FUNCTION "FC2039_ZC_TQ" : Void
TITLE = FC2038_TQ
{ S7_Optimized_Access := 'TRUE' }
AUTHOR : HCR
FAMILY : ZeusControl
VERSION : 1.0
//Funcion para gestion dispositivo tanque.
   VAR_INPUT
      Pulso1seg : Bool;
      Arranque : Bool;
   END_VAR

   VAR_TEMP
      for_i : Int;
      for_mux_cambios : Int;
      for_mux : Int;
      t_Index : Int;
      t_oldIndex : Int;
      t_NumLL : Int;
      t_NumHL : Int;
      t_NumBH : Int;
      t_NumNivel : Int;
      t_NumTemperatura : Int;
      t_x0 : Real;
      t_x1 : Real;
      t_x : Real;
      t_y0 : Real;
      t_y1 : Real;
      t_RadioCilindro : Real;
      t_RadioConoInf : Real;
      t_RadioActual : Real;
      t_Vol1 : Real;
      t_Vol2 : Real;
      t_Vol3 : Real;
      t_ConsignaAgitador : Real;
      t_AlarmaNivel : Bool;
      t_AlarmaTemperatura : Bool;
      t_VacioLL : Bool;
      t_VacioEA : Bool;
      t_AlarmaConfigD : Bool;
      t_AlarmaConfigEA : Bool;
      t_AlarmaConfigV : Bool;
      t_AlarmaConfigAG : Bool;
      t_HistPositiva : Real;
      t_HistNegativa : Real;
      t_ElseCase : Bool;
   END_VAR

   VAR CONSTANT
      CONSTANTE_EMPIRICA : Real := 10.1;
      CONSTANTE_PI : Real := 3.141593;
      ESTADO_DESHABILITADO : Int := 0;
      ESTADO_SUCIO : Int := 1;
      ESTADO_LIMPIO : Int := 2;
      ESTADO_PRODUCTO : Int := 3;
      ESTADO_CIP : Int := 4;
   END_VAR


BEGIN
	(*
	ZEUS CONTROL, S.A.
	(c)Copyright (2022) All Rights Reserved
	--------------------------------------------------------------------------------------

	Software:       TIA Portal 16
	Restricciones:  PLC serie 1200/1500

	Nombre:         DISPOSITIVO TANQUE
	Descripcion:    Modelo de dispositivo tanque

	Dependencias:
	    FC:         FC15025_ZC_CONTADOR_TIEMPO_V1_01
	    FB:         -
	    DB:         DB2018_DISP_TQ
	                DB1_SYS
	    UDT:        ZC_DISP_TQ
	                ZC_MUX
	                ZC_TON
	                ZC_CONTADOR_TIEMPO

	Change log:

	    Version     Fecha       Tecnico a cargo     Descripción

	    01.00.01    26.04.2022  (HCR)               Primera versión.
	    01.00.02    09.10.2023  (HCR)               Cambio en activacion dispositivos para que actue solamente cuando tenga producto.
	    01.00.03    15.04.2024  (ABH)               Se añade gestion multiplexado para Scada (no indexado)
	    01.00.04    08.01.2025  (ABH)               Se añade entrada de primer arranque del PLC para resetear indices de multiplexado
	                                                Se añade movimiento de TQ[0] a multiplexado en caso de que el indice sea 0.
	    01.00.05    24.01.2025  (ABH)               Se modifica la logica del multiplexado, la asignacion de oldindex se cambia de sitio ya que de vez en cuando (dependiendo de cuando el HMI
	                                                realiza la comunicacion asincrona con el PLC) no detectaba el cambio y se machacaban valores.
	    01.00.16    26.03.2025  (ABH)               Se añade variable grupo de alarma para separar los nuevos avisos por cuadro.
	    02.00.00    17.12.2025  (ABH)               Se eliminan los idiomas. Se utiliza codigos para trazabilidad. Se elimina entrada "Idioma". Se elimina nombre de UDT. Se añade indexHMI para lista de
	                                                texto en sistemas de supervision.

	//=====================================================================================
	*)

	REGION MULTIPLEXADO

	    //  ===========================================================================================================
	    //  Al arranque del PLC, ponemos a 0 todos los indices de los multiplexados y salimos del bloque sin gestionarlo
	    IF #Arranque THEN
	        FOR #for_mux := 0 TO "N_MAX_MUX_DISP" DO
	            "DB2039_TQ".Mux[#for_mux].Index :=
	            "DB2039_TQ".Mux[#for_mux].oldIndex := 0;
	        END_FOR;
	        RETURN;
	    END_IF;

	    //  ===========================================================================================================
	    //  Gestion de multiplexado
	    FOR #for_mux := 0 TO "N_MAX_MUX_DISP" DO

	        //  ===============================================================================================================
	        //  Antes de iniciar la logica del multiplexado, revisamos los limites
	        REGION LIMITES

	            //  ===========================================================================================================
	            //  Limites
	            IF "DB2039_TQ".Mux[#for_mux].Index < 0 THEN
	                "DB2039_TQ".Mux[#for_mux].Index := 0;
	            END_IF;
	            IF "DB2039_TQ".Mux[#for_mux].Index > "N_MAX_DISP_TQ" THEN
	                "DB2039_TQ".Mux[#for_mux].Index := "N_MAX_DISP_TQ";
	            END_IF;
	            IF "DB2039_TQ".Mux[#for_mux].Index >= "N_MAX_DISP_TQ" THEN
	                "DB2039_TQ".Mux[#for_mux].MaxVisible := TRUE;
	            ELSE
	                "DB2039_TQ".Mux[#for_mux].MaxVisible := FALSE;
	            END_IF;

	        END_REGION

	        //  Pasamos el indice a variable temporal para evisar cambios no deseados
	        #t_Index := "DB2039_TQ".Mux[#for_mux].Index;
	        #t_oldIndex := "DB2039_TQ".Mux[#for_mux].oldIndex;

	        //  ===========================================================================================================
	        //  Valor anterior del indice
	        "DB2039_TQ".Mux[#for_mux].oldIndex := #t_Index;

	        IF "DB2039_TQ".Mux[#for_mux].Habilitar THEN

	            //  ===========================================================================================================
	            //  Gestionamos solo los tipos
	            IF #t_Index > 0 THEN



	                REGION CARGA_INICIAL

	                    //  ===========================================================================================================
	                    //  Al detectar un cambio en el indice del dispositivo, cargamos los valores del dispositivo que tenga el indice.
	                    IF #t_Index <> #t_oldIndex THEN
	                        "DB2039_TQ".Mux[#for_mux].TQ := "DB2039_TQ".TQ[#t_Index];
	                    END_IF;

	                END_REGION



	                REGION DATOS_LECTURA

	                    //  ===========================================================================================================
	                    //  Movimiento de datos gestionados en FC
	                    "DB2039_TQ".Mux[#for_mux].TQ.Hmi_Index := "DB2039_TQ".TQ[#t_Index].Hmi_Index;
	                    "DB2039_TQ".Mux[#for_mux].TQ.Hmi_Estado := "DB2039_TQ".TQ[#t_Index].Hmi_Estado;
	                    "DB2039_TQ".Mux[#for_mux].TQ.Estado_TanqueVacio  := "DB2039_TQ".TQ[#t_Index].Estado_TanqueVacio;
	                    "DB2039_TQ".Mux[#for_mux].TQ.Estado_PocisionAltura  := "DB2039_TQ".TQ[#t_Index].Estado_PocisionAltura;
	                    "DB2039_TQ".Mux[#for_mux].TQ.Estado_NivelBajo  := "DB2039_TQ".TQ[#t_Index].Estado_NivelBajo;
	                    "DB2039_TQ".Mux[#for_mux].TQ.Estado_NivelAlto  := "DB2039_TQ".TQ[#t_Index].Estado_NivelAlto;
	                    "DB2039_TQ".Mux[#for_mux].TQ.Estado_BocaHombre  := "DB2039_TQ".TQ[#t_Index].Estado_BocaHombre;
	                    "DB2039_TQ".Mux[#for_mux].TQ.Estado_Mezcla  := "DB2039_TQ".TQ[#t_Index].Estado_Mezcla;
	                    "DB2039_TQ".Mux[#for_mux].TQ.Alarmas_NivelBajo  := "DB2039_TQ".TQ[#t_Index].Alarmas_NivelBajo;
	                    "DB2039_TQ".Mux[#for_mux].TQ.Alarmas_NivelAlto  := "DB2039_TQ".TQ[#t_Index].Alarmas_NivelAlto;
	                    "DB2039_TQ".Mux[#for_mux].TQ.Alarmas_BocaHombre  := "DB2039_TQ".TQ[#t_Index].Alarmas_BocaHombre;
	                    "DB2039_TQ".Mux[#for_mux].TQ.Alarmas_Instrumentacion  := "DB2039_TQ".TQ[#t_Index].Alarmas_Instrumentacion;
	                    "DB2039_TQ".Mux[#for_mux].TQ.Alarmas_Parametros  := "DB2039_TQ".TQ[#t_Index].Alarmas_Parametros;
	                    "DB2039_TQ".Mux[#for_mux].TQ.Alarmas_General  := "DB2039_TQ".TQ[#t_Index].Alarmas_General;
	                    "DB2039_TQ".Mux[#for_mux].TQ.Alarmas_Capacidad  := "DB2039_TQ".TQ[#t_Index].Alarmas_Capacidad;
	                    "DB2039_TQ".Mux[#for_mux].TQ.Aux_VisConsignaTemperatura  := "DB2039_TQ".TQ[#t_Index].Aux_VisConsignaTemperatura;
	                    "DB2039_TQ".Mux[#for_mux].TQ.Aux_PulsoAlternarAG  := "DB2039_TQ".TQ[#t_Index].Aux_PulsoAlternarAG;
	                    "DB2039_TQ".Mux[#for_mux].TQ.Aux_MemOrdenAgitador  := "DB2039_TQ".TQ[#t_Index].Aux_MemOrdenAgitador;
	                    "DB2039_TQ".Mux[#for_mux].TQ.Aux_MemOrdenTemperatura  := "DB2039_TQ".TQ[#t_Index].Aux_MemOrdenTemperatura;
	                    "DB2039_TQ".Mux[#for_mux].TQ.Aux_MemOrdenProducto  := "DB2039_TQ".TQ[#t_Index].Aux_MemOrdenProducto;
	                    "DB2039_TQ".Mux[#for_mux].TQ.Aux_MemEstadoCIP  := "DB2039_TQ".TQ[#t_Index].Aux_MemEstadoCIP;
	                    "DB2039_TQ".Mux[#for_mux].TQ.Aux_CipOK := "DB2039_TQ".TQ[#t_Index].Aux_CipOK;

	                    "DB2039_TQ".Mux[#for_mux].TQ.Orden_ParoControlAgitador := "DB2039_TQ".TQ[#t_Index].Orden_ParoControlAgitador;
	                    "DB2039_TQ".Mux[#for_mux].TQ.Orden_ParoControlTemp := "DB2039_TQ".TQ[#t_Index].Orden_ParoControlTemp;

	                    "DB2039_TQ".Mux[#for_mux].TQ.Estado_EA_Nivel  := "DB2039_TQ".TQ[#t_Index].Estado_EA_Nivel;
	                    "DB2039_TQ".Mux[#for_mux].TQ.Estado_EA_Temperatura  := "DB2039_TQ".TQ[#t_Index].Estado_EA_Temperatura;
	                    "DB2039_TQ".Mux[#for_mux].TQ.Estado_Tanque := "DB2039_TQ".TQ[#t_Index].Estado_Tanque;
	                    "DB2039_TQ".Mux[#for_mux].TQ.Estado_Producto1  := "DB2039_TQ".TQ[#t_Index].Estado_Producto1;
	                    "DB2039_TQ".Mux[#for_mux].TQ.Estado_Producto2  := "DB2039_TQ".TQ[#t_Index].Estado_Producto2;
	                    "DB2039_TQ".Mux[#for_mux].TQ.Estado_Volumen  := "DB2039_TQ".TQ[#t_Index].Estado_Volumen;
	                    "DB2039_TQ".Mux[#for_mux].TQ.Estado_Presion  := "DB2039_TQ".TQ[#t_Index].Estado_Presion;
	                    "DB2039_TQ".Mux[#for_mux].TQ.Estado_Altura  := "DB2039_TQ".TQ[#t_Index].Estado_Altura;

	                    "DB2039_TQ".Mux[#for_mux].TQ.Tiempos_TiempoProducto := "DB2039_TQ".TQ[#t_Index].Tiempos_TiempoProducto;
	                    "DB2039_TQ".Mux[#for_mux].TQ.Tiempos_TiempoLimpio := "DB2039_TQ".TQ[#t_Index].Tiempos_TiempoLimpio;
	                    "DB2039_TQ".Mux[#for_mux].TQ.Tiempos_RetTanqueVacio  := "DB2039_TQ".TQ[#t_Index].Tiempos_RetTanqueVacio;
	                    "DB2039_TQ".Mux[#for_mux].TQ.Tiempos_AgitadorONActual := "DB2039_TQ".TQ[#t_Index].Tiempos_AgitadorONActual;
	                    "DB2039_TQ".Mux[#for_mux].TQ.Tiempos_AgitadorOFFActual := "DB2039_TQ".TQ[#t_Index].Tiempos_AgitadorOFFActual;

	                    "DB2039_TQ".Mux[#for_mux].TQ.Config_HabilitarCalculoVol := "DB2039_TQ".TQ[#t_Index].Config_HabilitarCalculoVol;
	                    "DB2039_TQ".Mux[#for_mux].TQ.Config_HabilitarCamisa := "DB2039_TQ".TQ[#t_Index].Config_HabilitarCamisa;
	                    "DB2039_TQ".Mux[#for_mux].TQ.Config_HabilitarAlarmas := "DB2039_TQ".TQ[#t_Index].Config_HabilitarAlarmas;
	                    "DB2039_TQ".Mux[#for_mux].TQ.Config_HabilitarAgitador := "DB2039_TQ".TQ[#t_Index].Config_HabilitarAgitador;
	                    "DB2039_TQ".Mux[#for_mux].TQ.Config_GrupoAlarma := "DB2039_TQ".TQ[#t_Index].Config_GrupoAlarma;

	                    "DB2039_TQ".Mux[#for_mux].TQ.Aux_ValorTarjetaNivel  := "DB2039_TQ".TQ[#t_Index].Aux_ValorTarjetaNivel;
	                    "DB2039_TQ".Mux[#for_mux].TQ.Aux_ValorIngeneriaTemperatura  := "DB2039_TQ".TQ[#t_Index].Aux_ValorIngeneriaTemperatura;
	                    "DB2039_TQ".Mux[#for_mux].TQ.Orden_Temperatura := "DB2039_TQ".TQ[#t_Index].Orden_Temperatura;
	                    "DB2039_TQ".Mux[#for_mux].TQ.Orden_Agitacion := "DB2039_TQ".TQ[#t_Index].Orden_Agitacion;
	                    "DB2039_TQ".Mux[#for_mux].TQ.Orden_CIP := "DB2039_TQ".TQ[#t_Index].Orden_CIP;
	                    "DB2039_TQ".Mux[#for_mux].TQ.Orden_Producto := "DB2039_TQ".TQ[#t_Index].Orden_Producto;
	                    "DB2039_TQ".Mux[#for_mux].TQ.Orden_TipoProducto := "DB2039_TQ".TQ[#t_Index].Orden_TipoProducto;
	                    "DB2039_TQ".Mux[#for_mux].TQ.Orden_ConsignaAgitador := "DB2039_TQ".TQ[#t_Index].Orden_ConsignaAgitador;

	                END_REGION

	                REGION DATOS_ESCRITURA

	                    //  ===========================================================================================================
	                    //  Reinicializamos valor existe cambio
	                    "DB2039_TQ".Mux[#for_mux].ExisteCambio := false;

	                    //  ===========================================================================================================
	                    //  Ordenes
	                    IF "DB2039_TQ".Mux[#for_mux].TQ.Estado_TanqueNuevo <> "DB2039_TQ".TQ[#t_Index].Estado_TanqueNuevo THEN
	                        "DB2039_TQ".TQ[#t_Index].Estado_TanqueNuevo := "DB2039_TQ".Mux[#for_mux].TQ.Estado_TanqueNuevo;
	                        "DB2039_TQ".Mux[#for_mux].ExisteCambio := true;
	                    END_IF;
	                    IF "DB2039_TQ".Mux[#for_mux].TQ.Estado_ProductoNuevo <> "DB2039_TQ".TQ[#t_Index].Estado_ProductoNuevo THEN
	                        "DB2039_TQ".TQ[#t_Index].Estado_ProductoNuevo := "DB2039_TQ".Mux[#for_mux].TQ.Estado_ProductoNuevo;
	                        "DB2039_TQ".Mux[#for_mux].ExisteCambio := true;
	                    END_IF;
	                    IF "DB2039_TQ".Mux[#for_mux].TQ.Orden_CambioEstado <> "DB2039_TQ".TQ[#t_Index].Orden_CambioEstado THEN
	                        "DB2039_TQ".TQ[#t_Index].Orden_CambioEstado := "DB2039_TQ".Mux[#for_mux].TQ.Orden_CambioEstado;
	                        "DB2039_TQ".Mux[#for_mux].TQ.Orden_CambioEstado := FALSE;
	                        "DB2039_TQ".Mux[#for_mux].ExisteCambio := true;
	                     END_IF;
	                    IF "DB2039_TQ".Mux[#for_mux].TQ.Orden_CambioProd1 <> "DB2039_TQ".TQ[#t_Index].Orden_CambioProd1 THEN
	                        "DB2039_TQ".TQ[#t_Index].Orden_CambioProd1 := "DB2039_TQ".Mux[#for_mux].TQ.Orden_CambioProd1;
	                        "DB2039_TQ".Mux[#for_mux].TQ.Orden_CambioProd1 := FALSE;
	                        "DB2039_TQ".Mux[#for_mux].ExisteCambio := true;
	                    END_IF;
	                    IF "DB2039_TQ".Mux[#for_mux].TQ.Orden_CambioProd2 <> "DB2039_TQ".TQ[#t_Index].Orden_CambioProd2 THEN
	                        "DB2039_TQ".TQ[#t_Index].Orden_CambioProd2 := "DB2039_TQ".Mux[#for_mux].TQ.Orden_CambioProd2;
	                        "DB2039_TQ".Mux[#for_mux].TQ.Orden_CambioProd2 := FALSE;
	                        "DB2039_TQ".Mux[#for_mux].ExisteCambio := true;
	                    END_IF;

	                    //  ===========================================================================================================
	                    //  Configuracion
	                    IF "DB2039_TQ".Mux[#for_mux].TQ.Config_HabilitarControlAgitacion <> "DB2039_TQ".TQ[#t_Index].Config_HabilitarControlAgitacion THEN
	                        "DB2039_TQ".TQ[#t_Index].Config_HabilitarControlAgitacion := "DB2039_TQ".Mux[#for_mux].TQ.Config_HabilitarControlAgitacion;
	                        "DB2039_TQ".Mux[#for_mux].ExisteCambio := true;
	                    END_IF;
	                    IF "DB2039_TQ".Mux[#for_mux].TQ.Config_HabilitarControlTemp <> "DB2039_TQ".TQ[#t_Index].Config_HabilitarControlTemp THEN
	                        "DB2039_TQ".TQ[#t_Index].Config_HabilitarControlTemp := "DB2039_TQ".Mux[#for_mux].TQ.Config_HabilitarControlTemp;
	                        "DB2039_TQ".Mux[#for_mux].ExisteCambio := true;
	                     END_IF;
	                    IF "DB2039_TQ".Mux[#for_mux].TQ.Config_TipoControlTemperatura <> "DB2039_TQ".TQ[#t_Index].Config_TipoControlTemperatura THEN
	                        "DB2039_TQ".TQ[#t_Index].Config_TipoControlTemperatura := "DB2039_TQ".Mux[#for_mux].TQ.Config_TipoControlTemperatura;
	                        "DB2039_TQ".Mux[#for_mux].ExisteCambio := true;
	                    END_IF;
	                    IF "DB2039_TQ".Mux[#for_mux].TQ.Config_NumeroEANivel <> "DB2039_TQ".TQ[#t_Index].Config_NumeroEANivel THEN
	                        "DB2039_TQ".TQ[#t_Index].Config_NumeroEANivel := "DB2039_TQ".Mux[#for_mux].TQ.Config_NumeroEANivel;
	                        "DB2039_TQ".Mux[#for_mux].ExisteCambio := true;
	                     END_IF;
	                    IF "DB2039_TQ".Mux[#for_mux].TQ.Config_NumeroEATemp <> "DB2039_TQ".TQ[#t_Index].Config_NumeroEATemp THEN
	                        "DB2039_TQ".TQ[#t_Index].Config_NumeroEATemp := "DB2039_TQ".Mux[#for_mux].TQ.Config_NumeroEATemp;
	                        "DB2039_TQ".Mux[#for_mux].ExisteCambio := true;
	                    END_IF;
	                    IF "DB2039_TQ".Mux[#for_mux].TQ.Config_NumeroLL <> "DB2039_TQ".TQ[#t_Index].Config_NumeroLL THEN
	                        "DB2039_TQ".TQ[#t_Index].Config_NumeroLL := "DB2039_TQ".Mux[#for_mux].TQ.Config_NumeroLL;
	                        "DB2039_TQ".Mux[#for_mux].ExisteCambio := true;
	                    END_IF;
	                    IF "DB2039_TQ".Mux[#for_mux].TQ.Config_NumeroHL <> "DB2039_TQ".TQ[#t_Index].Config_NumeroHL THEN
	                        "DB2039_TQ".TQ[#t_Index].Config_NumeroHL := "DB2039_TQ".Mux[#for_mux].TQ.Config_NumeroHL;
	                        "DB2039_TQ".Mux[#for_mux].ExisteCambio := true;
	                    END_IF;
	                    IF "DB2039_TQ".Mux[#for_mux].TQ.Config_NumeroBH <> "DB2039_TQ".TQ[#t_Index].Config_NumeroBH THEN
	                        "DB2039_TQ".TQ[#t_Index].Config_NumeroBH := "DB2039_TQ".Mux[#for_mux].TQ.Config_NumeroBH;
	                        "DB2039_TQ".Mux[#for_mux].ExisteCambio := true;
	                     END_IF;
	                    IF "DB2039_TQ".Mux[#for_mux].TQ.Config_NumeroVA <> "DB2039_TQ".TQ[#t_Index].Config_NumeroVA THEN
	                        "DB2039_TQ".TQ[#t_Index].Config_NumeroVA := "DB2039_TQ".Mux[#for_mux].TQ.Config_NumeroVA;
	                        "DB2039_TQ".Mux[#for_mux].ExisteCambio := true;
	                     END_IF;
	                    IF "DB2039_TQ".Mux[#for_mux].TQ.Config_NumeroAG <> "DB2039_TQ".TQ[#t_Index].Config_NumeroAG THEN
	                        "DB2039_TQ".TQ[#t_Index].Config_NumeroAG := "DB2039_TQ".Mux[#for_mux].TQ.Config_NumeroAG;
	                        "DB2039_TQ".Mux[#for_mux].ExisteCambio := true;
	                     END_IF;
	                    IF "DB2039_TQ".Mux[#for_mux].TQ.Config_TipoAgitacionTiempo <> "DB2039_TQ".TQ[#t_Index].Config_TipoAgitacionTiempo THEN
	                        "DB2039_TQ".TQ[#t_Index].Config_TipoAgitacionTiempo := "DB2039_TQ".Mux[#for_mux].TQ.Config_TipoAgitacionTiempo;
	                        "DB2039_TQ".Mux[#for_mux].ExisteCambio := true;
	                     END_IF;
	                    IF "DB2039_TQ".Mux[#for_mux].TQ.Config_TipoAgitacionVelocidad <> "DB2039_TQ".TQ[#t_Index].Config_TipoAgitacionVelocidad THEN
	                        "DB2039_TQ".TQ[#t_Index].Config_TipoAgitacionVelocidad := "DB2039_TQ".Mux[#for_mux].TQ.Config_TipoAgitacionVelocidad;
	                        "DB2039_TQ".Mux[#for_mux].ExisteCambio := true;
	                    END_IF;
	                    IF "DB2039_TQ".Mux[#for_mux].TQ.Config_TipoAgitador <> "DB2039_TQ".TQ[#t_Index].Config_TipoAgitador THEN
	                        "DB2039_TQ".TQ[#t_Index].Config_TipoAgitador := "DB2039_TQ".Mux[#for_mux].TQ.Config_TipoAgitador;
	                        "DB2039_TQ".Mux[#for_mux].ExisteCambio := true;
	                    END_IF;
	                    IF "DB2039_TQ".Mux[#for_mux].TQ.Config_EscaladoMinTarjeta <> "DB2039_TQ".TQ[#t_Index].Config_EscaladoMinTarjeta THEN
	                        "DB2039_TQ".TQ[#t_Index].Config_EscaladoMinTarjeta := "DB2039_TQ".Mux[#for_mux].TQ.Config_EscaladoMinTarjeta;
	                        "DB2039_TQ".Mux[#for_mux].ExisteCambio := true;
	                    END_IF;
	                    IF "DB2039_TQ".Mux[#for_mux].TQ.Config_EscaladoMaxTarjeta <> "DB2039_TQ".TQ[#t_Index].Config_EscaladoMaxTarjeta THEN
	                        "DB2039_TQ".TQ[#t_Index].Config_EscaladoMaxTarjeta := "DB2039_TQ".Mux[#for_mux].TQ.Config_EscaladoMaxTarjeta;
	                        "DB2039_TQ".Mux[#for_mux].ExisteCambio := true;
	                     END_IF;
	                    IF "DB2039_TQ".Mux[#for_mux].TQ.Config_EscaladoMinIngenieria <> "DB2039_TQ".TQ[#t_Index].Config_EscaladoMinIngenieria THEN
	                        "DB2039_TQ".TQ[#t_Index].Config_EscaladoMinIngenieria := "DB2039_TQ".Mux[#for_mux].TQ.Config_EscaladoMinIngenieria;
	                        "DB2039_TQ".Mux[#for_mux].ExisteCambio := true;
	                     END_IF;
	                    IF "DB2039_TQ".Mux[#for_mux].TQ.Config_EscaladoMaxIngenieria <> "DB2039_TQ".TQ[#t_Index].Config_EscaladoMaxIngenieria THEN
	                        "DB2039_TQ".TQ[#t_Index].Config_EscaladoMaxIngenieria := "DB2039_TQ".Mux[#for_mux].TQ.Config_EscaladoMaxIngenieria;
	                        "DB2039_TQ".Mux[#for_mux].ExisteCambio := true;
	                     END_IF;
	                    IF "DB2039_TQ".Mux[#for_mux].TQ.Config_ConsignaTemperatura <> "DB2039_TQ".TQ[#t_Index].Config_ConsignaTemperatura THEN
	                        "DB2039_TQ".TQ[#t_Index].Config_ConsignaTemperatura := "DB2039_TQ".Mux[#for_mux].TQ.Config_ConsignaTemperatura;
	                        "DB2039_TQ".Mux[#for_mux].ExisteCambio := true;
	                     END_IF;
	                    IF "DB2039_TQ".Mux[#for_mux].TQ.Config_HisteresisTemperatura <> "DB2039_TQ".TQ[#t_Index].Config_HisteresisTemperatura THEN
	                        "DB2039_TQ".TQ[#t_Index].Config_HisteresisTemperatura := "DB2039_TQ".Mux[#for_mux].TQ.Config_HisteresisTemperatura;
	                        "DB2039_TQ".Mux[#for_mux].ExisteCambio := true;
	                    END_IF;
	                    IF "DB2039_TQ".Mux[#for_mux].TQ.Config_VolumenMinControlTemp <> "DB2039_TQ".TQ[#t_Index].Config_VolumenMinControlTemp THEN
	                        "DB2039_TQ".TQ[#t_Index].Config_VolumenMinControlTemp := "DB2039_TQ".Mux[#for_mux].TQ.Config_VolumenMinControlTemp;
	                        "DB2039_TQ".Mux[#for_mux].ExisteCambio := true;
	                    END_IF;
	                    IF "DB2039_TQ".Mux[#for_mux].TQ.Config_VolumenMaxControlTemp <> "DB2039_TQ".TQ[#t_Index].Config_VolumenMaxControlTemp THEN
	                        "DB2039_TQ".TQ[#t_Index].Config_VolumenMaxControlTemp := "DB2039_TQ".Mux[#for_mux].TQ.Config_VolumenMaxControlTemp;
	                        "DB2039_TQ".Mux[#for_mux].ExisteCambio := true;
	                    END_IF;
	                    IF "DB2039_TQ".Mux[#for_mux].TQ.Config_VolumenMinControlAgitador <> "DB2039_TQ".TQ[#t_Index].Config_VolumenMinControlAgitador THEN
	                        "DB2039_TQ".TQ[#t_Index].Config_VolumenMinControlAgitador := "DB2039_TQ".Mux[#for_mux].TQ.Config_VolumenMinControlAgitador;
	                        "DB2039_TQ".Mux[#for_mux].ExisteCambio := true;
	                    END_IF;
	                    IF "DB2039_TQ".Mux[#for_mux].TQ.Config_VolumenMaxControlAgitador <> "DB2039_TQ".TQ[#t_Index].Config_VolumenMaxControlAgitador THEN
	                        "DB2039_TQ".TQ[#t_Index].Config_VolumenMaxControlAgitador := "DB2039_TQ".Mux[#for_mux].TQ.Config_VolumenMaxControlAgitador;
	                        "DB2039_TQ".Mux[#for_mux].ExisteCambio := true;
	                    END_IF;
	                    IF "DB2039_TQ".Mux[#for_mux].TQ.Config_VolumenTanqueVacio <> "DB2039_TQ".TQ[#t_Index].Config_VolumenTanqueVacio THEN
	                        "DB2039_TQ".TQ[#t_Index].Config_VolumenTanqueVacio := "DB2039_TQ".Mux[#for_mux].TQ.Config_VolumenTanqueVacio;
	                        "DB2039_TQ".Mux[#for_mux].ExisteCambio := true;
	                    END_IF;
	                    IF "DB2039_TQ".Mux[#for_mux].TQ.Config_VelocidadMinAgitador <> "DB2039_TQ".TQ[#t_Index].Config_VelocidadMinAgitador THEN
	                        "DB2039_TQ".TQ[#t_Index].Config_VelocidadMinAgitador := "DB2039_TQ".Mux[#for_mux].TQ.Config_VelocidadMinAgitador;
	                        "DB2039_TQ".Mux[#for_mux].ExisteCambio := true;
	                    END_IF;
	                    IF "DB2039_TQ".Mux[#for_mux].TQ.Config_VelocidadMaxAgitador <> "DB2039_TQ".TQ[#t_Index].Config_VelocidadMaxAgitador THEN
	                        "DB2039_TQ".TQ[#t_Index].Config_VelocidadMaxAgitador := "DB2039_TQ".Mux[#for_mux].TQ.Config_VelocidadMaxAgitador;
	                        "DB2039_TQ".Mux[#for_mux].ExisteCambio := true;
	                    END_IF;
	                    IF "DB2039_TQ".Mux[#for_mux].TQ.Config_VelocidadFijaAgitador <> "DB2039_TQ".TQ[#t_Index].Config_VelocidadFijaAgitador THEN
	                        "DB2039_TQ".TQ[#t_Index].Config_VelocidadFijaAgitador := "DB2039_TQ".Mux[#for_mux].TQ.Config_VelocidadFijaAgitador;
	                        "DB2039_TQ".Mux[#for_mux].ExisteCambio := true;
	                    END_IF;
	                    IF "DB2039_TQ".Mux[#for_mux].TQ.Config_CapacidadTanque <> "DB2039_TQ".TQ[#t_Index].Config_CapacidadTanque THEN
	                        "DB2039_TQ".TQ[#t_Index].Config_CapacidadTanque := "DB2039_TQ".Mux[#for_mux].TQ.Config_CapacidadTanque;
	                        "DB2039_TQ".Mux[#for_mux].ExisteCambio := true;
	                    END_IF;
	                    IF "DB2039_TQ".Mux[#for_mux].TQ.Config_DiametroCilindro <> "DB2039_TQ".TQ[#t_Index].Config_DiametroCilindro THEN
	                        "DB2039_TQ".TQ[#t_Index].Config_DiametroCilindro := "DB2039_TQ".Mux[#for_mux].TQ.Config_DiametroCilindro;
	                        "DB2039_TQ".Mux[#for_mux].ExisteCambio := true;
	                    END_IF;
	                    IF "DB2039_TQ".Mux[#for_mux].TQ.Config_AlturaCilindro <> "DB2039_TQ".TQ[#t_Index].Config_AlturaCilindro THEN
	                        "DB2039_TQ".TQ[#t_Index].Config_AlturaCilindro := "DB2039_TQ".Mux[#for_mux].TQ.Config_AlturaCilindro;
	                        "DB2039_TQ".Mux[#for_mux].ExisteCambio := true;
	                    END_IF;
	                    IF "DB2039_TQ".Mux[#for_mux].TQ.Config_DiametroConoInferior <> "DB2039_TQ".TQ[#t_Index].Config_DiametroConoInferior THEN
	                        "DB2039_TQ".TQ[#t_Index].Config_DiametroConoInferior := "DB2039_TQ".Mux[#for_mux].TQ.Config_DiametroConoInferior;
	                        "DB2039_TQ".Mux[#for_mux].ExisteCambio := true;
	                    END_IF;
	                    IF "DB2039_TQ".Mux[#for_mux].TQ.Config_AnguloCono <> "DB2039_TQ".TQ[#t_Index].Config_AnguloCono THEN
	                        "DB2039_TQ".TQ[#t_Index].Config_AnguloCono := "DB2039_TQ".Mux[#for_mux].TQ.Config_AnguloCono;
	                        "DB2039_TQ".Mux[#for_mux].ExisteCambio := true;
	                    END_IF;
	                    IF "DB2039_TQ".Mux[#for_mux].TQ.Config_AlturaCono <> "DB2039_TQ".TQ[#t_Index].Config_AlturaCono THEN
	                        "DB2039_TQ".TQ[#t_Index].Config_AlturaCono := "DB2039_TQ".Mux[#for_mux].TQ.Config_AlturaCono;
	                        "DB2039_TQ".Mux[#for_mux].ExisteCambio := true;
	                    END_IF;

	                    //  ===========================================================================================================
	                    //  Tiempos
	                    IF "DB2039_TQ".Mux[#for_mux].TQ.Tiempos_AgitadorONConsigna <> "DB2039_TQ".TQ[#t_Index].Tiempos_AgitadorONConsigna THEN
	                        "DB2039_TQ".TQ[#t_Index].Tiempos_AgitadorONConsigna := "DB2039_TQ".Mux[#for_mux].TQ.Tiempos_AgitadorONConsigna;
	                        "DB2039_TQ".Mux[#for_mux].ExisteCambio := true;
	                    END_IF;
	                    IF "DB2039_TQ".Mux[#for_mux].TQ.Tiempos_AgitadorOFFConsigna <> "DB2039_TQ".TQ[#t_Index].Tiempos_AgitadorOFFConsigna THEN
	                        "DB2039_TQ".TQ[#t_Index].Tiempos_AgitadorOFFConsigna := "DB2039_TQ".Mux[#for_mux].TQ.Tiempos_AgitadorOFFConsigna;
	                        "DB2039_TQ".Mux[#for_mux].ExisteCambio := true;
	                    END_IF;


	                END_REGION

	                REGION GESTION_CAMBIOS

	                    //  ===========================================================================================================
	                    //  Si existe cambios en el dispositivo generados por SCADA, actualizamos los datos en el resto de multiplexados,
	                    //  en caso de que este abierto el mismo dispositivo.
	                    IF "DB2039_TQ".Mux[#for_mux].ExisteCambio THEN
	                        //  Recorremos todos los multiplexados
	                        FOR #for_mux_cambios := 0 TO "N_MAX_MUX_DISP" DO

	                            //  No miramos el multiplexado actual
	                            IF #for_mux_cambios <> #for_mux THEN

	                                //  En caso de que este seleccionado el mismo indice, movemos el dispositivo al multiplexado
	                                //  correspondiente
	                                IF #t_Index = "DB2039_TQ".Mux[#for_mux_cambios].Index THEN
	                                    "DB2039_TQ".Mux[#for_mux_cambios].TQ := "DB2039_TQ".TQ[#t_Index];
	                                END_IF;

	                            END_IF;

	                        END_FOR;
	                        "DB2039_TQ".Mux[#for_mux].ExisteCambio := FALSE;
	                    END_IF;

	                END_REGION

	            ELSE

	                //  ===========================================================================================================
	                //  En caso de que el indice sea 0, movemos el valor de la EA[0] que no se usa para escribir el index.
	                "DB2039_TQ".Mux[#for_mux].TQ := "DB2039_TQ".TQ[0];

	            END_IF;

	        ELSE

	            "DB2039_TQ".Mux[#for_mux].ExisteCambio := FALSE;
	            "DB2039_TQ".Mux[#for_mux].Index :=
	            "DB2039_TQ".Mux[#for_mux].oldIndex := 0;

	        END_IF;

	    END_FOR;

	END_REGION

	REGION LOGICA_DEL_DISPOSITIVO

	    // =============================================================================
	    // Resetear todas las alarmas para que se vuelvan a generar
	    FOR #for_i := 0 TO "N_MAX_DISP_AGRUP" DO
	        "DB2039_TQ".Agrup[#for_i].AlgunaAlarma := FALSE;
	        "DB2039_TQ".Agrup[#for_i].AlgunaEnManual := FALSE;
	    END_FOR;

	    FOR #for_i := 1 TO "N_MAX_DISP_TQ" DO

	        "DB2039_TQ".TQ[#t_Index].Hmi_Index := #for_i + "DISP_OFFSET_TQ";

	        // =============================================================================
	        //  CAMBIO DE ESTADO DESDE HMI/SCADA
	        IF "DB2039_TQ".TQ[#for_i].Orden_CambioEstado THEN
	            "DB2039_TQ".TQ[#for_i].Estado_Tanque := "DB2039_TQ".TQ[#for_i].Estado_TanqueNuevo;
	            "DB2039_TQ".TQ[#for_i].Orden_CambioEstado := FALSE;
	        END_IF;


	        "DB2039_TQ".TQ[#for_i].Config_Habilitar := ("DB2039_TQ".TQ[#for_i].Estado_Tanque <> #ESTADO_DESHABILITADO);

	        // =============================================================================
	        // DISPOSITIVO HABILITADO
	        // =============================================================================
	        IF "DB2039_TQ".TQ[#for_i].Config_Habilitar THEN

	            REGION LIMITE_GRUPO_ALARMA

	                IF "DB2039_TQ".TQ[#for_i].Config_GrupoAlarma < 0 THEN
	                    "DB2039_TQ".TQ[#for_i].Config_GrupoAlarma := 0;
	                END_IF;
	                IF "DB2039_TQ".TQ[#for_i].Config_GrupoAlarma > "N_MAX_DISP_AGRUP" THEN
	                    "DB2039_TQ".TQ[#for_i].Config_GrupoAlarma := "N_MAX_DISP_AGRUP";
	                END_IF;

	            END_REGION

	            REGION ASIGNAR_DISPOSITIVOS

	                // =============================================================================
	                //  ASIGNACION DISPOSITOS
	                #t_NumLL := "DB2039_TQ".TQ[#for_i].Config_NumeroLL;
	                #t_NumHL := "DB2039_TQ".TQ[#for_i].Config_NumeroHL;
	                #t_NumBH := "DB2039_TQ".TQ[#for_i].Config_NumeroBH;
	                #t_NumNivel := "DB2039_TQ".TQ[#for_i].Config_NumeroEANivel;
	                #t_NumTemperatura := "DB2039_TQ".TQ[#for_i].Config_NumeroEATemp;
	                // =============================================================================
	                //  DETECTOR BOCA DE HOMBRE
	                IF #t_NumBH > 0 AND #t_NumBH <= "N_MAX_DISP_ED" THEN
	                    "DB2039_TQ".TQ[#for_i].Estado_BocaHombre := "DB2000_ED".ED[#t_NumBH].Estado_Activado;
	                END_IF;
	                // =============================================================================
	                //  DETECTOR LL
	                IF #t_NumLL > 0 AND #t_NumLL <= "N_MAX_DISP_ED" THEN
	                    "DB2039_TQ".TQ[#for_i].Estado_NivelBajo := "DB2000_ED".ED[#t_NumLL].Estado_Activado;
	                END_IF;
	                // =============================================================================
	                //  DETECTOR HL
	                IF #t_NumHL > 0 AND #t_NumHL <= "N_MAX_DISP_ED" THEN
	                    "DB2039_TQ".TQ[#for_i].Estado_NivelAlto := "DB2000_ED".ED[#t_NumHL].Estado_Activado;
	                END_IF;
	                // =============================================================================
	                //  LECTURA VALOR TARJETA NIVEL
	                IF #t_NumNivel > 0 AND #t_NumNivel <= "N_MAX_DISP_EA" THEN
	                    "DB2039_TQ".TQ[#for_i].Aux_ValorTarjetaNivel := "DB2001_EA".EA[#t_NumNivel].Estado_ValorTarjeta;
	                END_IF;
	                // =============================================================================
	                //  LECTURA VALOR INGENERIA TEMPERATURA
	                IF #t_NumTemperatura > 0 AND #t_NumTemperatura <= "N_MAX_DISP_EA" THEN
	                    "DB2039_TQ".TQ[#for_i].Aux_ValorIngeneriaTemperatura := "DB2001_EA".EA[#t_NumTemperatura].Estado_ValorIngenieria;
	                END_IF;

	            END_REGION

	            REGION ALARMAS
	                // =============================================================================
	                //  ALARMA CONFIGURACIÓN
	                #t_AlarmaConfigD := ("DB2039_TQ".TQ[#for_i].Config_NumeroBH > "N_MAX_DISP_ED") OR ("DB2039_TQ".TQ[#for_i].Config_NumeroLL > "N_MAX_DISP_ED") OR ("DB2039_TQ".TQ[#for_i].Config_NumeroHL > "N_MAX_DISP_ED");
	                #t_AlarmaConfigEA := ("DB2039_TQ".TQ[#for_i].Config_NumeroEANivel > "N_MAX_DISP_EA") OR ("DB2039_TQ".TQ[#for_i].Config_NumeroEATemp > "N_MAX_DISP_EA");
	                #t_AlarmaConfigV := "DB2039_TQ".TQ[#for_i].Config_HabilitarCamisa AND "DB2039_TQ".TQ[#for_i].Config_NumeroVA > "N_MAX_DISP_V";

	                IF "DB2039_TQ".TQ[#for_i].Config_HabilitarAgitador THEN
	                    CASE "DB2039_TQ".TQ[#for_i].Config_TipoAgitador OF
	                        0:  // Motor
	                            #t_AlarmaConfigAG := "DB2039_TQ".TQ[#for_i].Config_NumeroAG > "N_MAX_DISP_M";
	                        1:  // VF
	                            #t_AlarmaConfigAG := "DB2039_TQ".TQ[#for_i].Config_NumeroAG > "N_MAX_DISP_M_VF";
	                            ;
	                        2:  // SINA
	                            #t_AlarmaConfigAG := "DB2039_TQ".TQ[#for_i].Config_NumeroAG > "N_MAX_DISP_M_SINA";
	                        ELSE  // Statement section ELSE
	                            #t_AlarmaConfigAG := TRUE;
	                    END_CASE;
	                END_IF;

	                "DB2039_TQ".TQ[#for_i].Alarmas_Parametros := #t_AlarmaConfigD OR #t_AlarmaConfigEA OR #t_AlarmaConfigV OR #t_AlarmaConfigAG;

	                IF "DB2039_TQ".TQ[#for_i].Config_HabilitarAlarmas THEN
	                    // =============================================================================
	                    //  ALARMA DETECTOR NIVEL MÍNIMO
	                    IF #t_NumLL > 0 AND #t_NumLL <= "N_MAX_DISP_ED" THEN
	                        "DB2039_TQ".TQ[#for_i].Alarmas_NivelBajo := NOT "DB2039_TQ".TQ[#for_i].Estado_NivelBajo;
	                    ELSE
	                        "DB2039_TQ".TQ[#for_i].Alarmas_NivelBajo := FALSE;
	                    END_IF;
	                    // =============================================================================
	                    //  ALARMA DETECTOR NIVEL MÁXIMO
	                    IF #t_NumHL > 0 AND #t_NumHL <= "N_MAX_DISP_ED" THEN
	                        "DB2039_TQ".TQ[#for_i].Alarmas_NivelAlto := "DB2039_TQ".TQ[#for_i].Estado_NivelAlto;
	                    ELSE
	                        "DB2039_TQ".TQ[#for_i].Alarmas_NivelAlto := FALSE;
	                    END_IF;
	                    // =============================================================================
	                    //  ALARMA DETECTOR BOCA HOMBRE
	                    IF #t_NumBH > 0 AND #t_NumBH <= "N_MAX_DISP_ED" THEN
	                        "DB2039_TQ".TQ[#for_i].Alarmas_BocaHombre := NOT "DB2039_TQ".TQ[#for_i].Estado_BocaHombre;
	                    ELSE
	                        "DB2039_TQ".TQ[#for_i].Alarmas_BocaHombre := FALSE;
	                    END_IF;
	                    // =============================================================================
	                    //  ALARMA DE INSTRUMENTACIÓN
	                    IF #t_NumNivel > 0 AND #t_NumNivel <= "N_MAX_DISP_EA" THEN
	                        #t_AlarmaNivel := ("DB2001_EA".EA[#t_NumNivel].Aux_Estado = 6 OR
	                        "DB2001_EA".EA[#t_NumNivel].Aux_Estado = 3 OR
	                        "DB2001_EA".EA[#t_NumNivel].Aux_Estado = 4 OR
	                        "DB2001_EA".EA[#t_NumNivel].Aux_Estado = 5 OR
	                        "DB2001_EA".EA[#t_NumNivel].Aux_Estado = 7 OR
	                        "DB2001_EA".EA[#t_NumNivel].Aux_Estado = 8);
	                    ELSE
	                        #t_AlarmaNivel := FALSE;
	                    END_IF;

	                    IF #t_NumTemperatura > 0 AND #t_NumTemperatura <= "N_MAX_DISP_EA" THEN
	                        #t_AlarmaTemperatura := ("DB2001_EA".EA[#t_NumNivel].Aux_Estado = 6 OR
	                        "DB2001_EA".EA[#t_NumTemperatura].Aux_Estado = 3 OR
	                        "DB2001_EA".EA[#t_NumTemperatura].Aux_Estado = 4 OR
	                        "DB2001_EA".EA[#t_NumTemperatura].Aux_Estado = 5 OR
	                        "DB2001_EA".EA[#t_NumTemperatura].Aux_Estado = 7 OR
	                        "DB2001_EA".EA[#t_NumTemperatura].Aux_Estado = 8);
	                    ELSE
	                        #t_AlarmaTemperatura := FALSE;
	                    END_IF;

	                    "DB2039_TQ".TQ[#for_i].Alarmas_Instrumentacion := #t_AlarmaNivel OR #t_AlarmaTemperatura OR
	                    ("DB2039_TQ".TQ[#for_i].Config_EscaladoMinIngenieria >= "DB2039_TQ".TQ[#for_i].Config_EscaladoMaxIngenieria) OR
	                    ("DB2039_TQ".TQ[#for_i].Config_EscaladoMinTarjeta >= "DB2039_TQ".TQ[#for_i].Config_EscaladoMaxTarjeta);

	                    // =============================================================================
	                    //  ALARMA POR CAPACIDAD
	                    "DB2039_TQ".TQ[#for_i].Alarmas_Capacidad := "DB2039_TQ".TQ[#for_i].Estado_Volumen > "DB2039_TQ".TQ[#for_i].Config_CapacidadTanque;

	                    // =============================================================================
	                    //  ALARMA GENERAL
	                    "DB2039_TQ".TQ[#for_i].Alarmas_General := "DB2039_TQ".TQ[#for_i].Alarmas_NivelBajo OR
	                    "DB2039_TQ".TQ[#for_i].Alarmas_NivelAlto OR
	                    "DB2039_TQ".TQ[#for_i].Alarmas_BocaHombre OR
	                    "DB2039_TQ".TQ[#for_i].Alarmas_Instrumentacion OR
	                    "DB2039_TQ".TQ[#for_i].Alarmas_Capacidad;

	                ELSE
	                    "DB2039_TQ".TQ[#for_i].Alarmas_General := FALSE;
	                    "DB2039_TQ".TQ[#for_i].Alarmas_NivelBajo := FALSE;
	                    "DB2039_TQ".TQ[#for_i].Alarmas_NivelAlto := FALSE;
	                    "DB2039_TQ".TQ[#for_i].Alarmas_BocaHombre := FALSE;
	                    "DB2039_TQ".TQ[#for_i].Alarmas_Instrumentacion := FALSE;
	                    "DB2039_TQ".TQ[#for_i].Alarmas_Capacidad := FALSE;
	                END_IF;
	            END_REGION

	            REGION VOLUMEN

	                REGION ESTADO VOLUMEN

	                    "DB2039_TQ".TQ[#for_i].Estado_EA_Nivel := 1;  //  Estado normal

	                    IF #t_NumNivel > 0 AND
	                        (("DB2039_TQ".TQ[#for_i].Config_EscaladoMaxIngenieria = "DB2039_TQ".TQ[#for_i].Config_EscaladoMinIngenieria) OR
	                        ("DB2039_TQ".TQ[#for_i].Config_EscaladoMaxTarjeta = "DB2039_TQ".TQ[#for_i].Config_EscaladoMinTarjeta) OR
	                        ("DB2001_EA".EA[#t_NumNivel].Aux_Estado = 6)) THEN
	                        "DB2039_TQ".TQ[#for_i].Estado_EA_Nivel := 6; //  Error de configuración
	                    END_IF;

	                    IF #t_NumNivel > 0 AND
	                        (("DB2039_TQ".TQ[#for_i].Config_EscaladoMaxIngenieria < "DB2039_TQ".TQ[#for_i].Config_EscaladoMinIngenieria) OR
	                        ("DB2039_TQ".TQ[#for_i].Config_EscaladoMaxTarjeta < "DB2039_TQ".TQ[#for_i].Config_EscaladoMinTarjeta) OR
	                        ("DB2001_EA".EA[#t_NumNivel].Aux_Estado = 6)) THEN
	                        "DB2039_TQ".TQ[#for_i].Estado_EA_Nivel := 6; //  Error de configuración
	                    END_IF;

	                    IF "DB2001_EA".EA[#t_NumNivel].Aux_Estado = 3 THEN
	                        "DB2039_TQ".TQ[#for_i].Estado_EA_Nivel := 3; //  Error de canal
	                    END_IF;

	                    IF "DB2001_EA".EA[#t_NumNivel].Aux_Estado = 4 THEN
	                        "DB2039_TQ".TQ[#for_i].Estado_EA_Nivel := 4; //  Volumen en alarma
	                    END_IF;

	                    IF "DB2001_EA".EA[#t_NumNivel].Aux_Estado = 5 THEN
	                        "DB2039_TQ".TQ[#for_i].Estado_EA_Nivel := 5; //  Volumen en alarma
	                    END_IF;

	                    IF "DB2001_EA".EA[#t_NumNivel].Aux_Estado = 7 THEN
	                        "DB2039_TQ".TQ[#for_i].Estado_EA_Nivel := 7; //  Error de lectura
	                    END_IF;

	                    IF "DB2001_EA".EA[#t_NumNivel].Aux_Estado = 8 THEN
	                        "DB2039_TQ".TQ[#for_i].Estado_EA_Nivel := 8; //  EA no direccionada
	                    END_IF;

	                    IF "DB2001_EA".EA[#t_NumNivel].Estado_AutoMan THEN
	                        "DB2039_TQ".TQ[#for_i].Estado_EA_Nivel := 2; //  Señal forzada
	                    END_IF;

	                    IF ("DB2001_EA".EA[#t_NumNivel].Aux_Estado = 0) OR (#t_NumNivel = 0) THEN
	                        "DB2039_TQ".TQ[#for_i].Estado_EA_Nivel := 0; //  Señal deshabilitada
	                    END_IF;

	                    // =============================================================================
	                    //  POSICIÓN DE ALTURA
	                    //  0 - Altura en cono, 1 - Altura por encima del cono
	                    "DB2039_TQ".TQ[#for_i].Estado_PocisionAltura := ("DB2039_TQ".TQ[#for_i].Estado_Altura > "DB2039_TQ".TQ[#for_i].Config_AlturaCono) AND (#t_NumNivel > 0);

	                    // =============================================================================
	                    //  TANQUE VACÍO
	                    #t_VacioLL := (NOT "DB2039_TQ".TQ[#for_i].Estado_NivelBajo) AND (#t_NumLL > 0);
	                    // =============================================================================
	                    //  GESTION TON PARA EA < VOLUMEN TANQUE VACIO
	                    //"DB2039_TQ".TQ[#for_i].Tiempos_RetTanqueVacio.SP := 10;
	                    "DB2039_TQ".TQ[#for_i].Tiempos_RetTanqueVacio.SP := 25;
	                    "DB2039_TQ".TQ[#for_i].Tiempos_RetTanqueVacio.IN := ("DB2039_TQ".TQ[#for_i].Estado_Volumen < "DB2039_TQ".TQ[#for_i].Config_VolumenTanqueVacio) AND (#t_NumNivel > 0);
	                    IF "DB2039_TQ".TQ[#for_i].Tiempos_RetTanqueVacio.IN THEN
	                        IF "DB2039_TQ".TQ[#for_i].Tiempos_RetTanqueVacio.ET >= "DB2039_TQ".TQ[#for_i].Tiempos_RetTanqueVacio.SP THEN
	                            "DB2039_TQ".TQ[#for_i].Tiempos_RetTanqueVacio.Q := TRUE;
	                        ELSE
	                            IF #Pulso1seg THEN
	                                "DB2039_TQ".TQ[#for_i].Tiempos_RetTanqueVacio.ET += 1;
	                            END_IF;
	                        END_IF;
	                    ELSE
	                        "DB2039_TQ".TQ[#for_i].Tiempos_RetTanqueVacio.ET := 0;
	                        "DB2039_TQ".TQ[#for_i].Tiempos_RetTanqueVacio.Q := FALSE;
	                    END_IF;
	                    #t_VacioEA := "DB2039_TQ".TQ[#for_i].Tiempos_RetTanqueVacio.Q;
	                    "DB2039_TQ".TQ[#for_i].Estado_TanqueVacio := #t_VacioLL OR #t_VacioEA;

	                END_REGION

	                REGION CALCULO_VOLUMEN_TANQUE

	                    // =============================================================================
	                    // HABILITADO CALCULO DE VOLUMEN
	                    IF "DB2039_TQ".TQ[#for_i].Config_HabilitarCalculoVol THEN

	                        // =============================================================================
	                        //  VALORES DE ESCALADO
	                        #t_x0 := INT_TO_REAL("DB2039_TQ".TQ[#for_i].Config_EscaladoMinTarjeta);
	                        #t_x1 := INT_TO_REAL("DB2039_TQ".TQ[#for_i].Config_EscaladoMaxTarjeta);
	                        #t_x := DINT_TO_REAL("DB2039_TQ".TQ[#for_i].Aux_ValorTarjetaNivel);
	                        #t_y0 := "DB2039_TQ".TQ[#for_i].Config_EscaladoMinIngenieria;
	                        #t_y1 := "DB2039_TQ".TQ[#for_i].Config_EscaladoMaxIngenieria;

	                        // =============================================================================
	                        // SEÑAL EN ESTADO CORRECTO
	                        IF "DB2039_TQ".TQ[#for_i].Estado_EA_Nivel <> 6 AND
	                            "DB2039_TQ".TQ[#for_i].Estado_EA_Nivel <> 3 AND
	                            "DB2039_TQ".TQ[#for_i].Estado_EA_Nivel <> 7 AND
	                            "DB2039_TQ".TQ[#for_i].Estado_EA_Nivel <> 8 THEN

	                            // =============================================================================
	                            // SEÑAL EN AUTOMATICO
	                            IF NOT "DB2001_EA".EA[#t_NumNivel].Estado_AutoMan THEN

	                                // =============================================================================
	                                // ESCALADO
	                                "DB2039_TQ".TQ[#for_i].Estado_Presion := (((#t_x - #t_x0) * ((#t_y1 - #t_y0) / (#t_x1 - #t_x0))) + #t_y0);
	                                // =============================================================================
	                                // LÍMITE MAX
	                                IF "DB2039_TQ".TQ[#for_i].Estado_Presion > "DB2039_TQ".TQ[#for_i].Config_EscaladoMaxIngenieria THEN
	                                    "DB2039_TQ".TQ[#for_i].Estado_Presion := "DB2039_TQ".TQ[#for_i].Config_EscaladoMaxIngenieria;
	                                END_IF;
	                                // =============================================================================
	                                // LÍMITE MIN
	                                IF "DB2039_TQ".TQ[#for_i].Estado_Presion < "DB2039_TQ".TQ[#for_i].Config_EscaladoMinIngenieria THEN
	                                    "DB2039_TQ".TQ[#for_i].Estado_Presion := "DB2039_TQ".TQ[#for_i].Config_EscaladoMinIngenieria;
	                                END_IF;

	                                // =============================================================================
	                                // CÁLCULO DE COLUMNA DE LÍQUIDO
	                                "DB2039_TQ".TQ[#for_i].Estado_Altura := "DB2039_TQ".TQ[#for_i].Estado_Presion * #CONSTANTE_EMPIRICA;
	                                //PENDIENTE VER SI ES NECESARIO LIMITAR CON LA COLUMAN DEL CILINDRO **************************************

	                                // =============================================================================
	                                // CÁLCULO DE DIMENSIONES
	                                #t_RadioCilindro := "DB2039_TQ".TQ[#for_i].Config_DiametroCilindro / 2.0;
	                                #t_RadioConoInf := "DB2039_TQ".TQ[#for_i].Config_DiametroConoInferior / 2.0;
	                                #t_RadioActual := #t_RadioCilindro;

	                                // =============================================================================
	                                // ALTURA INFERIOR AL CONO
	                                IF "DB2039_TQ".TQ[#for_i].Estado_Altura < "DB2039_TQ".TQ[#for_i].Config_AlturaCono THEN
	                                    #t_RadioActual := ("DB2039_TQ".TQ[#for_i].Estado_Altura / TAN("DB2039_TQ".TQ[#for_i].Config_AnguloCono)); //+0.13
	                                    // =============================================================================
	                                    // LÍMITE RADIO
	                                    IF #t_RadioActual > #t_RadioCilindro THEN
	                                        #t_RadioActual := #t_RadioCilindro;
	                                    END_IF;

	                                    // =============================================================================
	                                    // CÁLCULO DE VOLUMEN INFERIOR AL CONO
	                                    IF "DB2039_TQ".TQ[#for_i].Estado_Altura > 0 THEN
	                                        #t_Vol1 := (#t_RadioConoInf * #t_RadioConoInf) + (#t_RadioActual * #t_RadioActual) + (#t_RadioConoInf * #t_RadioActual);
	                                        #t_Vol2 := (#CONSTANTE_PI * "DB2039_TQ".TQ[#for_i].Estado_Altura) / 3.0;
	                                        "DB2039_TQ".TQ[#for_i].Estado_Volumen := #t_Vol1 * #t_Vol2 * 1000.0;
	                                    ELSE
	                                        "DB2039_TQ".TQ[#for_i].Estado_Volumen := 0.0;
	                                    END_IF;
	                                    // =============================================================================
	                                    // ALTURA SUPERIOR AL CONO
	                                ELSE
	                                    #t_Vol1 := (#t_RadioConoInf * #t_RadioConoInf) + (#t_RadioActual * #t_RadioActual) + (#t_RadioConoInf * #t_RadioActual);
	                                    #t_Vol2 := (#CONSTANTE_PI * "DB2039_TQ".TQ[#for_i].Estado_Altura) / 3.0;
	                                    #t_Vol3 := #CONSTANTE_PI * #t_RadioCilindro * #t_RadioCilindro * ("DB2039_TQ".TQ[#for_i].Estado_Altura - "DB2039_TQ".TQ[#for_i].Config_AlturaCono);
	                                    "DB2039_TQ".TQ[#for_i].Estado_Volumen := ((#t_Vol1 * #t_Vol2) + #t_Vol3) * 1000.0;
	                                END_IF;
	                            ELSE
	                                // =============================================================================
	                                // ESTADO MANUAL DE EA DE NIVEL
	                                "DB2039_TQ".TQ[#for_i].Estado_Volumen := "DB2001_EA".EA[#t_NumNivel].Orden_ConsignaManual;
	                            END_IF;

	                        ELSE
	                            "DB2039_TQ".TQ[#for_i].Estado_Volumen := 0.0;
	                        END_IF;


	                    ELSE

	                        "DB2039_TQ".TQ[#for_i].Estado_Volumen := "DB2001_EA".EA[#t_NumNivel].Estado_ValorIngenieria;

	                    END_IF;

	                END_REGION

	            END_REGION

	            REGION TEMPERATURA

	                REGION ESTADO_TEMPERATURA

	                    "DB2039_TQ".TQ[#for_i].Estado_EA_Temperatura := 1;  //  Estado normal

	                    IF #t_NumTemperatura > 0 AND ("DB2001_EA".EA[#t_NumTemperatura].Aux_Estado = 6) THEN
	                        "DB2039_TQ".TQ[#for_i].Estado_EA_Temperatura := 6; //  Error de configuración
	                    END_IF;

	                    IF "DB2001_EA".EA[#t_NumTemperatura].Aux_Estado = 3 THEN
	                        "DB2039_TQ".TQ[#for_i].Estado_EA_Temperatura := 3; //  Error de canal
	                    END_IF;

	                    IF "DB2001_EA".EA[#t_NumTemperatura].Aux_Estado = 4 THEN
	                        "DB2039_TQ".TQ[#for_i].Estado_EA_Temperatura := 4; //  Volumen en alarma
	                    END_IF;

	                    IF "DB2001_EA".EA[#t_NumTemperatura].Aux_Estado = 5 THEN
	                        "DB2039_TQ".TQ[#for_i].Estado_EA_Temperatura := 5; //  Volumen en alarma
	                    END_IF;

	                    IF "DB2001_EA".EA[#t_NumTemperatura].Aux_Estado = 7 THEN
	                        "DB2039_TQ".TQ[#for_i].Estado_EA_Temperatura := 7; //  Error de lectura
	                    END_IF;

	                    IF "DB2001_EA".EA[#t_NumTemperatura].Aux_Estado = 8 THEN
	                        "DB2039_TQ".TQ[#for_i].Estado_EA_Temperatura := 8; //  EA no direccionada
	                    END_IF;

	                    IF "DB2001_EA".EA[#t_NumTemperatura].Estado_AutoMan THEN
	                        "DB2039_TQ".TQ[#for_i].Estado_EA_Temperatura := 2; //  Señal forzada
	                    END_IF;

	                    IF ("DB2001_EA".EA[#t_NumTemperatura].Aux_Estado = 0) OR (#t_NumNivel = 0) THEN
	                        "DB2039_TQ".TQ[#for_i].Estado_EA_Temperatura := 0; //  Señal deshabilitada
	                    END_IF;

	                END_REGION

	            END_REGION

	            REGION ESTADO

	                // =============================================================================
	                //  ESTADO SUCIO
	                IF "DB2039_TQ".TQ[#for_i].Estado_Tanque = #ESTADO_PRODUCTO AND "DB2039_TQ".TQ[#for_i].Estado_TanqueVacio AND "DB2039_TQ".TQ[#for_i].Estado_ComOk THEN
	                    "DB2039_TQ".TQ[#for_i].Estado_Tanque := #ESTADO_SUCIO;
	                END_IF;

	                // =============================================================================
	                //  ESTADO CIP
	                IF "DB2039_TQ".TQ[#for_i].Orden_CIP AND NOT "DB2039_TQ".TQ[#for_i].Aux_MemEstadoCIP THEN
	                    "DB2039_TQ".TQ[#for_i].Estado_Tanque := #ESTADO_CIP;
	                    "DB2039_TQ".TQ[#for_i].Aux_MemEstadoCIP := "DB2039_TQ".TQ[#for_i].Orden_CIP;
	                END_IF;

	                // =============================================================================
	                //  ESTADO LIMPIO
	                IF NOT "DB2039_TQ".TQ[#for_i].Orden_CIP AND "DB2039_TQ".TQ[#for_i].Aux_MemEstadoCIP THEN
	                    IF "DB2039_TQ".TQ[#for_i].Aux_CipOK THEN
	                        "DB2039_TQ".TQ[#for_i].Estado_Tanque := #ESTADO_LIMPIO;
	                    END_IF;
	                    "DB2039_TQ".TQ[#for_i].Aux_MemEstadoCIP := "DB2039_TQ".TQ[#for_i].Orden_CIP;
	                END_IF;

	                IF "DB2039_TQ".TQ[#for_i].Estado_Tanque = #ESTADO_CIP AND NOT "DB2039_TQ".TQ[#for_i].Orden_CIP AND NOT "DB2039_TQ".TQ[#for_i].Aux_CipOK THEN
	                    "DB2039_TQ".TQ[#for_i].Estado_Tanque := #ESTADO_SUCIO;
	                    "DB2039_TQ".TQ[#for_i].Aux_MemEstadoCIP := "DB2039_TQ".TQ[#for_i].Orden_CIP;
	                END_IF;

	                //  CONTADOR TIEMPO LIMPIO
	                "FC15025_ZC_CONTADOR_TIEMPO"(Pulso1seg := #Pulso1seg,
	                                             Iniciar := "DB2039_TQ".TQ[#for_i].Estado_Tanque = #ESTADO_LIMPIO,
	                                             Reset := "DB2039_TQ".TQ[#for_i].Estado_Tanque <> #ESTADO_LIMPIO,
	                                             Contador := "DB2039_TQ".TQ[#for_i].Tiempos_TiempoLimpio);

	                // =============================================================================
	                //  ESTADO PRODUCTO
	                IF "DB2039_TQ".TQ[#for_i].Orden_Producto AND NOT "DB2039_TQ".TQ[#for_i].Estado_TanqueVacio THEN
	                    "DB2039_TQ".TQ[#for_i].Estado_Tanque := #ESTADO_PRODUCTO;
	                END_IF;


	                // =============================================================================
	                //  CAMBIO DE ESTADO DESDE HMI/SCADA
	                IF "DB2039_TQ".TQ[#for_i].Orden_CambioProd1 THEN
	                    "DB2039_TQ".TQ[#for_i].Estado_Producto1 := "DB2039_TQ".TQ[#for_i].Estado_ProductoNuevo;
	                    "DB2039_TQ".TQ[#for_i].Orden_CambioProd1 := FALSE;
	                END_IF;
	                IF "DB2039_TQ".TQ[#for_i].Orden_CambioProd2 THEN
	                    "DB2039_TQ".TQ[#for_i].Estado_Producto2 := "DB2039_TQ".TQ[#for_i].Estado_ProductoNuevo;

	                    "DB2039_TQ".TQ[#for_i].Orden_CambioProd2 := FALSE;
	                END_IF;


	                // =============================================================================
	                //  PRODUCTOS
	                IF ("DB2039_TQ".TQ[#for_i].Estado_Tanque = #ESTADO_PRODUCTO) THEN
	                    IF "DB2039_TQ".TQ[#for_i].Orden_Producto AND NOT "DB2039_TQ".TQ[#for_i].Aux_MemOrdenProducto THEN
	                        IF "DB2039_TQ".TQ[#for_i].Estado_Producto2 = 0 AND "DB2039_TQ".TQ[#for_i].Estado_Producto1 <> 0 THEN
	                            "DB2039_TQ".TQ[#for_i].Estado_Producto2 := "DB2039_TQ".TQ[#for_i].Orden_TipoProducto;
	                        END_IF;
	                        IF "DB2039_TQ".TQ[#for_i].Estado_Producto1 = 0 THEN
	                            "DB2039_TQ".TQ[#for_i].Estado_Producto1 := "DB2039_TQ".TQ[#for_i].Orden_TipoProducto;
	                        END_IF;
	                    END_IF;
	                END_IF;
	                "DB2039_TQ".TQ[#for_i].Aux_MemOrdenProducto := "DB2039_TQ".TQ[#for_i].Orden_Producto;

	                IF NOT "DB2039_TQ".TQ[#for_i].Orden_Producto OR NOT ("DB2039_TQ".TQ[#for_i].Estado_Tanque = #ESTADO_PRODUCTO) THEN
	                    "DB2039_TQ".TQ[#for_i].Aux_MemOrdenProducto := FALSE;
	                END_IF;

	                "DB2039_TQ".TQ[#for_i].Orden_Producto := FALSE;

	                //  CONTADOR TIEMPO PRODUCTO
	                "FC15025_ZC_CONTADOR_TIEMPO"(Pulso1seg := #Pulso1seg,
	                                             Iniciar := "DB2039_TQ".TQ[#for_i].Estado_Tanque = #ESTADO_PRODUCTO,
	                                             Reset := "DB2039_TQ".TQ[#for_i].Estado_Tanque <> #ESTADO_PRODUCTO,
	                                             Contador := "DB2039_TQ".TQ[#for_i].Tiempos_TiempoProducto);

	                // =============================================================================
	                //  TANQUE MEZCLA
	                "DB2039_TQ".TQ[#for_i].Estado_Mezcla := "DB2039_TQ".TQ[#for_i].Estado_Producto1 <> 0 AND "DB2039_TQ".TQ[#for_i].Estado_Producto2 <> 0 AND "DB2039_TQ".TQ[#for_i].Estado_Producto1 <> "DB2039_TQ".TQ[#for_i].Estado_Producto2;

	                // =============================================================================
	                //  BORRADO DE PRODUCTOS
	                IF "DB2039_TQ".TQ[#for_i].Estado_Tanque <> #ESTADO_PRODUCTO THEN
	                    "DB2039_TQ".TQ[#for_i].Estado_Producto1 := 0;
	                    "DB2039_TQ".TQ[#for_i].Estado_Producto2 := 0;
	                END_IF;

	            END_REGION

	            REGION AGITADOR
	                // =============================================================================
	                // TANQUE CON AGITADOR
	                IF "DB2039_TQ".TQ[#for_i].Config_HabilitarAgitador AND NOT "DB2039_TQ".TQ[#for_i].Orden_ParoControlAgitador THEN

	                    // =============================================================================
	                    // HABILITAR AGITADOR
	                    IF "DB2039_TQ".TQ[#for_i].Config_HabilitarControlAgitacion THEN
	                        // =============================================================================
	                        // SE AÑADE 50 LITROS POR ENCIMA PARA EMPEZAR A AGITAR
	                        IF "DB2039_TQ".TQ[#for_i].Estado_Volumen > "DB2039_TQ".TQ[#for_i].Config_VolumenMinControlAgitador + 50.0 THEN
	                            "DB2039_TQ".TQ[#for_i].Aux_MemOrdenAgitador := TRUE;
	                            // =============================================================================
	                            //TIPO DE AGITACIÓN POR TIEMPO
	                            IF "DB2039_TQ".TQ[#for_i].Config_TipoAgitacionTiempo = 1 THEN
	                                // =============================================================================
	                                //TIEMPO ON DE AGITACIÓN
	                                IF #Pulso1seg AND "DB2039_TQ".TQ[#for_i].Aux_PulsoAlternarAG THEN
	                                    "DB2039_TQ".TQ[#for_i].Tiempos_AgitadorONActual += 1;
	                                END_IF;
	                                // =============================================================================
	                                //TIEMPO OFF DE AGITACIÓN
	                                IF #Pulso1seg AND NOT "DB2039_TQ".TQ[#for_i].Aux_PulsoAlternarAG THEN
	                                    "DB2039_TQ".TQ[#for_i].Tiempos_AgitadorOFFActual += 1;
	                                END_IF;
	                                // =============================================================================
	                                //CAMBIO DE ESTADO
	                                IF "DB2039_TQ".TQ[#for_i].Tiempos_AgitadorONActual >= "DB2039_TQ".TQ[#for_i].Tiempos_AgitadorONConsigna THEN
	                                    "DB2039_TQ".TQ[#for_i].Aux_PulsoAlternarAG := FALSE;
	                                    "DB2039_TQ".TQ[#for_i].Tiempos_AgitadorONActual := 0;
	                                END_IF;

	                                IF "DB2039_TQ".TQ[#for_i].Tiempos_AgitadorOFFActual >= "DB2039_TQ".TQ[#for_i].Tiempos_AgitadorOFFConsigna THEN
	                                    "DB2039_TQ".TQ[#for_i].Aux_PulsoAlternarAG := TRUE;
	                                    "DB2039_TQ".TQ[#for_i].Tiempos_AgitadorOFFActual := 0;
	                                END_IF;
	                            ELSE
	                                // =============================================================================
	                                //TIPO DE AGITACIÓN FIJO
	                                "DB2039_TQ".TQ[#for_i].Aux_PulsoAlternarAG := TRUE;
	                                "DB2039_TQ".TQ[#for_i].Tiempos_AgitadorOFFActual := 0;
	                                "DB2039_TQ".TQ[#for_i].Tiempos_AgitadorONActual := 0;
	                            END_IF;

	                            // =============================================================================
	                            //ORDEN ACTIVAR AGITADOR
	                            "DB2039_TQ".TQ[#for_i].Orden_Agitacion :=
	                            "DB2039_TQ".TQ[#for_i].Aux_PulsoAlternarAG AND
	                            ("DB2039_TQ".TQ[#for_i].Estado_BocaHombre OR "DB2039_TQ".TQ[#for_i].Config_NumeroBH = 0);

	                            // =============================================================================
	                            //FRECUENCIA DE AGITADOR
	                            IF "DB2039_TQ".TQ[#for_i].Orden_Agitacion AND "DB2039_TQ".TQ[#for_i].Config_TipoAgitador <> 0 THEN

	                                IF "DB2039_TQ".TQ[#for_i].Config_TipoAgitacionVelocidad = 0 THEN
	                                    // =============================================================================
	                                    //VELOCIDAD FIJA

	                                    "DB2039_TQ".TQ[#for_i].Orden_ConsignaAgitador := "DB2039_TQ".TQ[#for_i].Config_VelocidadFijaAgitador;

	                                ELSE
	                                    // =============================================================================
	                                    //VELOCIDAD POR NIVEL
	                                    #t_x0 := "DB2039_TQ".TQ[#for_i].Config_VolumenMinControlAgitador;
	                                    #t_x1 := "DB2039_TQ".TQ[#for_i].Config_VolumenMaxControlAgitador;
	                                    #t_x := "DB2039_TQ".TQ[#for_i].Estado_Volumen;
	                                    #t_y0 := "DB2039_TQ".TQ[#for_i].Config_VelocidadMinAgitador;
	                                    #t_y1 := "DB2039_TQ".TQ[#for_i].Config_VelocidadMaxAgitador;
	                                    #t_ConsignaAgitador := #t_y0 + (#t_y1 - #t_y0) * ((#t_x - #t_x0) / (#t_x1 - #t_x0));
	                                    IF #t_ConsignaAgitador > #t_y1 THEN
	                                        #t_ConsignaAgitador := #t_y1;
	                                    END_IF;
	                                    IF #t_ConsignaAgitador < #t_y0 THEN
	                                        #t_ConsignaAgitador := #t_y0;
	                                    END_IF;
	                                    "DB2039_TQ".TQ[#for_i].Orden_ConsignaAgitador := #t_ConsignaAgitador;
	                                END_IF;
	                            ELSE
	                                "DB2039_TQ".TQ[#for_i].Orden_ConsignaAgitador := 0.0;

	                            END_IF;

	                        END_IF;

	                        // =============================================================================
	                        //PARO AGITACIÓN POR NIVEL
	                        IF "DB2039_TQ".TQ[#for_i].Aux_MemOrdenAgitador AND "DB2039_TQ".TQ[#for_i].Estado_Volumen < "DB2039_TQ".TQ[#for_i].Config_VolumenMinControlAgitador - 20.0 THEN
	                            "DB2039_TQ".TQ[#for_i].Orden_Agitacion := FALSE;
	                            "DB2039_TQ".TQ[#for_i].Orden_ConsignaAgitador := 0.0;
	                            "DB2039_TQ".TQ[#for_i].Aux_PulsoAlternarAG := TRUE;
	                            "DB2039_TQ".TQ[#for_i].Aux_MemOrdenAgitador := FALSE;
	                            "DB2039_TQ".TQ[#for_i].Tiempos_AgitadorOFFActual := 0;
	                            "DB2039_TQ".TQ[#for_i].Tiempos_AgitadorONActual := 0;
	                        END_IF;

	                    ELSE
	                        "DB2039_TQ".TQ[#for_i].Config_HabilitarControlAgitacion := FALSE;
	                        "DB2039_TQ".TQ[#for_i].Orden_Agitacion := FALSE;
	                        "DB2039_TQ".TQ[#for_i].Orden_ConsignaAgitador := 0.0;
	                        "DB2039_TQ".TQ[#for_i].Aux_PulsoAlternarAG := TRUE;
	                        "DB2039_TQ".TQ[#for_i].Aux_MemOrdenAgitador := FALSE;
	                        "DB2039_TQ".TQ[#for_i].Tiempos_AgitadorOFFActual := 0;
	                        "DB2039_TQ".TQ[#for_i].Tiempos_AgitadorONActual := 0;
	                    END_IF;
	                END_IF;
	            END_REGION

	            REGION VALVULA

	                // =============================================================================
	                // TANQUE CON CONTROL DE TEMPERATURA
	                IF "DB2039_TQ".TQ[#for_i].Config_HabilitarCamisa AND NOT "DB2039_TQ".TQ[#for_i].Orden_ParoControlTemp THEN

	                #t_HistPositiva := "DB2039_TQ".TQ[#for_i].Config_ConsignaTemperatura + "DB2039_TQ".TQ[#for_i].Config_HisteresisTemperatura;
	                #t_HistNegativa := "DB2039_TQ".TQ[#for_i].Config_ConsignaTemperatura - "DB2039_TQ".TQ[#for_i].Config_HisteresisTemperatura;
	                    // =============================================================================
	                    // HABILITAR CONTROL DE TEMPERATURA
	                IF "DB2039_TQ".TQ[#for_i].Config_HabilitarControlTemp THEN

	                    IF "DB2039_TQ".TQ[#for_i].Estado_Volumen > "DB2039_TQ".TQ[#for_i].Config_VolumenMinControlTemp + 50.0 THEN
	                        "DB2039_TQ".TQ[#for_i].Aux_MemOrdenTemperatura := TRUE;
	                            // =============================================================================
	                            // CONTROL DE TEMPERATURA ENFRIAR
	                            IF "DB2039_TQ".TQ[#for_i].Config_TipoControlTemperatura THEN

	                                IF "DB2001_EA".EA[#t_NumTemperatura].Estado_ValorIngenieria > "DB2039_TQ".TQ[#for_i].Config_ConsignaTemperatura THEN
	                                    "DB2039_TQ".TQ[#for_i].Orden_Temperatura := TRUE;
	                                END_IF;

	                                IF "DB2001_EA".EA[#t_NumTemperatura].Estado_ValorIngenieria < #t_HistNegativa THEN
	                                    "DB2039_TQ".TQ[#for_i].Orden_Temperatura := FALSE;
	                                END_IF;
	                                // =============================================================================
	                                // CONTROL DE TEMPERATURA CALENTAR
	                            ELSE

	                                IF "DB2001_EA".EA[#t_NumTemperatura].Estado_ValorIngenieria < "DB2039_TQ".TQ[#for_i].Config_ConsignaTemperatura THEN
	                                    "DB2039_TQ".TQ[#for_i].Orden_Temperatura := TRUE;
	                                END_IF;

	                                IF "DB2001_EA".EA[#t_NumTemperatura].Estado_ValorIngenieria > #t_HistPositiva THEN
	                                    "DB2039_TQ".TQ[#for_i].Orden_Temperatura := FALSE;
	                                END_IF;

	                            END_IF;
	                        END_IF;
	                        // =============================================================================
	                        //PARAO CONTROL DE TEMPERATURA POR NIVEL
	                        IF "DB2039_TQ".TQ[#for_i].Aux_MemOrdenTemperatura AND "DB2039_TQ".TQ[#for_i].Estado_Volumen < "DB2039_TQ".TQ[#for_i].Config_VolumenMinControlTemp - 10.0 THEN
	                            "DB2039_TQ".TQ[#for_i].Orden_Temperatura := FALSE;
	                            "DB2039_TQ".TQ[#for_i].Aux_MemOrdenTemperatura := FALSE;
	                        END_IF;

	                    ELSE
	                        "DB2039_TQ".TQ[#for_i].Orden_Temperatura := FALSE;
	                    END_IF;


	                ELSE
	                    "DB2039_TQ".TQ[#for_i].Orden_Temperatura := FALSE;
	                END_IF;
	            END_REGION



	        ELSE
	            // =============================================================================
	            //  DISPOSITIVO DESHABILITADO
	            "DB2039_TQ".TQ[#for_i].Orden_Temperatura := FALSE;
	            "DB2039_TQ".TQ[#for_i].Orden_Agitacion := FALSE;
	            "DB2039_TQ".TQ[#for_i].Orden_ConsignaAgitador := 0.0;
	            "DB2039_TQ".TQ[#for_i].Orden_CIP := FALSE;
	            "DB2039_TQ".TQ[#for_i].Orden_Producto := FALSE;

	            "DB2039_TQ".TQ[#for_i].Orden_CambioEstado := FALSE;
	            "DB2039_TQ".TQ[#for_i].Orden_CambioProd1 := FALSE;
	            "DB2039_TQ".TQ[#for_i].Orden_CambioProd2 := FALSE;

	            "DB2039_TQ".TQ[#for_i].Aux_MemEstadoCIP := FALSE;
	            "DB2039_TQ".TQ[#for_i].Aux_MemOrdenProducto := FALSE;
	            "DB2039_TQ".TQ[#for_i].Aux_MemOrdenTemperatura := FALSE;
	            "DB2039_TQ".TQ[#for_i].Aux_MemOrdenAgitador := FALSE;

	            "DB2039_TQ".TQ[#for_i].Estado_TanqueVacio := FALSE;
	            "DB2039_TQ".TQ[#for_i].Estado_PocisionAltura := FALSE;
	            "DB2039_TQ".TQ[#for_i].Estado_NivelBajo := FALSE;
	            "DB2039_TQ".TQ[#for_i].Estado_NivelAlto := FALSE;
	            "DB2039_TQ".TQ[#for_i].Estado_BocaHombre := FALSE;

	            "DB2039_TQ".TQ[#for_i].Estado_Tanque := 0;  //  Deshabilitado
	            "DB2039_TQ".TQ[#for_i].Estado_Producto1 := 0;
	            "DB2039_TQ".TQ[#for_i].Estado_Producto2 := 0;



	            "DB2039_TQ".TQ[#for_i].Alarmas_NivelBajo := FALSE;
	            "DB2039_TQ".TQ[#for_i].Alarmas_NivelAlto := FALSE;
	            "DB2039_TQ".TQ[#for_i].Alarmas_BocaHombre:= FALSE;
	            "DB2039_TQ".TQ[#for_i].Alarmas_Capacidad := FALSE;
	            "DB2039_TQ".TQ[#for_i].Alarmas_Instrumentacion := FALSE;
	            "DB2039_TQ".TQ[#for_i].Alarmas_Parametros := FALSE;
	            "DB2039_TQ".TQ[#for_i].Alarmas_General := FALSE;

	            "DB2039_TQ".TQ[#for_i].Estado_Volumen := 0.0;
	            "DB2039_TQ".TQ[#for_i].Estado_Presion := 0.0;
	            "DB2039_TQ".TQ[#for_i].Estado_Altura := 0.0;

	            "DB2039_TQ".TQ[#for_i].Config_HabilitarControlAgitacion := FALSE;
	            "DB2039_TQ".TQ[#for_i].Config_HabilitarControlTemp := FALSE;

	            "DB2039_TQ".TQ[#for_i].Tiempos_AgitadorONActual := 0;
	            "DB2039_TQ".TQ[#for_i].Tiempos_AgitadorOFFActual := 0;
	            "DB2039_TQ".TQ[#for_i].Tiempos_RetTanqueVacio.ET := 0;
	            "DB2039_TQ".TQ[#for_i].Tiempos_RetTanqueVacio.Q := FALSE;

	            "DB2039_TQ".TQ[#for_i].Orden_ParoControlAgitador := FALSE;
	            "DB2039_TQ".TQ[#for_i].Orden_ParoControlTemp := FALSE;

	        END_IF;

	        REGION ACTIVAR DISPOSITIVOS

	            // =============================================================================
	            //  VISIBILIDAD CONSIGNA DE TEMPERATURA
	            "DB2039_TQ".TQ[#for_i].Aux_VisConsignaTemperatura :=
	            "DB2039_TQ".TQ[#for_i].Config_HabilitarCamisa AND
	            "DB2039_TQ".TQ[#for_i].Config_HabilitarControlTemp AND
	            "DB2039_TQ".TQ[#for_i].Aux_MemOrdenTemperatura AND
	            NOT "DB2039_TQ".TQ[#for_i].Orden_CIP AND ("DB2039_TQ".TQ[#for_i].Estado_Tanque = #ESTADO_PRODUCTO) AND
	            NOT "DB2039_TQ".TQ[#for_i].Orden_ParoControlTemp;

	            // =============================================================================
	            //  VÁLVULA DE CONTROL DE TEMPERATURA
	            IF NOT "DB2039_TQ".TQ[#for_i].Orden_CIP AND ("DB2039_TQ".TQ[#for_i].Estado_Tanque = #ESTADO_PRODUCTO) AND "DB2039_TQ".TQ[#for_i].Orden_Temperatura THEN
	                "DB2010_V".V["DB2039_TQ".TQ[#for_i].Config_NumeroVA].Orden_ActivarAuto := TRUE;
	            END_IF;

	            // =============================================================================
	            //  AGITADOR
	            CASE "DB2039_TQ".TQ[#for_i].Config_TipoAgitador OF
	                0:  // Motor
	                    IF NOT "DB2039_TQ".TQ[#for_i].Orden_CIP AND ("DB2039_TQ".TQ[#for_i].Estado_Tanque = #ESTADO_PRODUCTO) AND "DB2039_TQ".TQ[#for_i].Orden_Agitacion THEN
	                        "DB2015_M".M["DB2039_TQ".TQ[#for_i].Config_NumeroAG].Orden_ActivarAuto := TRUE;
	                    END_IF;
	                1:  // VF
	                    IF NOT "DB2039_TQ".TQ[#for_i].Orden_CIP AND ("DB2039_TQ".TQ[#for_i].Estado_Tanque = #ESTADO_PRODUCTO) AND "DB2039_TQ".TQ[#for_i].Orden_Agitacion THEN
	                        "DB2016_M_VF".M_VF["DB2039_TQ".TQ[#for_i].Config_NumeroAG].Orden_ActivarAuto := TRUE;
	                        "DB2016_M_VF".M_VF["DB2039_TQ".TQ[#for_i].Config_NumeroAG].Orden_ConsignaAuto := "DB2039_TQ".TQ[#for_i].Orden_ConsignaAgitador;
	                    END_IF;
	                2:  // SINA
	                    (* "DB2017_M_SINA".SINA["DB2039_TQ".TQ[#for_i].Config_NumeroAG].Orden.ActivarAuto := NOT "DB2039_TQ".TQ[#for_i].Orden_CIP AND ("DB2039_TQ".TQ[#for_i].Estado_Tanque = #PRODUCTO) AND "DB2039_TQ".TQ[#for_i].Orden_Agitacion;
	                    "DB2017_M_SINA".SINA["DB2039_TQ".TQ[#for_i].Config_NumeroAG].Orden.ConsignaAuto := "DB2039_TQ".TQ[#for_i].Orden_ConsignaAgitador; *)
	                    IF NOT "DB2039_TQ".TQ[#for_i].Orden_CIP AND ("DB2039_TQ".TQ[#for_i].Estado_Tanque = #ESTADO_PRODUCTO) AND "DB2039_TQ".TQ[#for_i].Orden_Agitacion THEN
	                        "DB2017_M_SINA".M_SINA["DB2039_TQ".TQ[#for_i].Config_NumeroAG].Orden_ActivarAuto := TRUE;
	                        "DB2016_M_VF".M_VF["DB2039_TQ".TQ[#for_i].Config_NumeroAG].Orden_ConsignaAuto := "DB2039_TQ".TQ[#for_i].Orden_ConsignaAgitador;
	                    END_IF;
	                    ;
	            END_CASE;

	        END_REGION

	        "DB2039_TQ".TQ[#for_i].Orden_ParoControlAgitador := FALSE;
	        "DB2039_TQ".TQ[#for_i].Orden_ParoControlTemp := FALSE;

	    END_FOR;

	END_REGION
END_FUNCTION

